{attribute 'GeneratedUsingTerminal: KL6211-0020'}
{attribute addProperty BoxType "KL6211-0020"}
{attribute addProperty Id "Channel_1AT %Q*Channel_099BCCDA0"}
{attribute addProperty CRC "2598716342"}
{attribute addProperty Size "0"}
TYPE KL_9AE543B6 :
STRUCT
	{attribute addProperty Name "Channel_1"}
	Channel_1 : Channel_099BCCDA;
END_STRUCT
END_TYPE

(* stored: Version 1.2.0.0, ProductVersion 3.1.4024.9
   DUT KL_9AE543B6: Id {8d673b33-e2f0-4a8e-8369-8fa4e5ae0b0a} *)
